PROGRAM MAIN
VAR
  _send : BOOL; // boolean, which can be triggered to send a message
  _openWeatherMapClient : OpenWeatherMap.OpenWeatherMapClient('<your_token>');   
END_VAR

IF _send
THEN
  _send := FALSE;
  _openWeatherMapClient.RequestWeatherByZipCodeAsync('6020', 'AT');
END_IF

_openWeatherMapClient.Cyclic();

END_PROGRAM

(* stored: Version 1.1.0.1, ProductVersion 3.1.4024.12
   POU MAIN: Id {33b3b19c-906c-4ad0-afd2-e113619d9985}, SpecialFunc None *)
